Staubli VAL3: cmdFaultReset.pgx

public program cmdFaultReset(num x_nAxNum)
begin
  //错误复位，'Fault reset'置1
  doFaultReset[x_nAxNum]=true
  delay(0.008)
  doFaultReset[x_nAxNum]=false
end
